// TwinCAT 3 PLC project Tc3_Element
// Title: Tc3_Element
// Company: Zerlauth
// Author: Peter Zerlauth
// ProjectVersion: 0.0.0.1
// Description: State Model with Observer and Events
// ProgramVersion: 3.1.4026.14
// CompilerDefines: release
// libraries:
//   Tc2_Standard, * (Beckhoff Automation GmbH)
//   Tc2_System, * (Beckhoff Automation GmbH)
//   Tc2_Utilities, * (Beckhoff Automation GmbH)
//   Tc3_Module,3.4.5.0,Beckhoff Automation GmbH
// project tree:
//   Element/Event/ E_Event.TcDUT, FB_Event.TcPOU, I_Event.TcIO, ST_Event.TcDUT (not stored), ST_EventFlags.TcDUT (not stored)
//   Element/Event/Observer/ FB_Observable.TcPOU (not stored), I_Observer.TcIO (not stored), I_Observable.TcIO (not stored)
//   Element/ E_Request.TcDUT, E_State.TcDUT, FB_Element.TcPOU, I_Element.TcIO (not stored)
//   Element/Reflection/ FB_Reflection.TcPOU (not stored), I_Reflection.TcIO
//   Element/Sequence/ E_Sequence.TcDUT (not stored), FB_Sequence.TcPOU (not stored), I_Sequence.TcIO (not stored), ST_Sequence.TcDUT (not stored), ST_SequenceOptions.TcDUT (not stored)
//   Level/ FB_Level.TcPOU
//   List/ FB_ListElement.TcPOU (not stored), FB_ListObject.TcPOU (not stored), FB_ListString.TcPOU (not stored), I_ListBase.TcIO (not stored), I_ListElement.TcIO (not stored), I_ListObject.TcIO (not stored), I_ListString.TcIO (not stored)
//   Logger/ FB_FileLogger.TcPOU, FB_LoggingProvider.TcPOU (not stored), FB_Logger.TcPOU, I_Logger.TcIO (not stored)
//   Module/ E_Mode.TcDUT (not stored), FB_Module.TcPOU, I_Module.TcIO (not stored)
//   Object/ FB_Object.TcPOU (not stored), I_Object.TcIO (not stored)
//   Utils/ FB_Debounce.TcPOU (not stored)
//   Utils/File/ FB_File.TcPOU, I_File.TcIO (not stored)
//   Version/ Global_Version.TcGVL (not stored)
// (motion and I/O tree: see PLC project development)
// real-time tasks:
//   TASK PlcTask: cycle T#500ms, priority 21, ADS port 351
//   TASK UnitTestTask: cycle T#1ms, priority 1, ADS port 350
// variable links:

// ---- Element/Event/E_Event.TcDUT
{attribute 'qualified_only'}
{attribute 'strict'}
{attribute 'to_string'}
TYPE E_Event :
(
	Verbose			:= 0,
	Debug			:= 1,
	Information		:= 2,
	Warning			:= 3,
	Error			:= 4
);
END_TYPE

// ---- Element/E_Request.TcDUT
{attribute 'qualified_only'}
{attribute 'strict'}
{attribute 'to_string'}

TYPE E_Request :
(
	{attribute 'analysis' := '-27'}
	Reset       := 1,
	{attribute 'analysis' := '-27'}
    Start       := 2,
	{attribute 'analysis' := '-27'}
	Stop		:= 3,
	{attribute 'analysis' := '-27'}
	Abort		:= 4
);
END_TYPE

// ---- Element/E_State.TcDUT
{attribute 'qualified_only'}
{attribute 'strict'}
{attribute 'to_string'}
TYPE E_State :
(
    Resetting       := 0,
   	Idle            := 1,
    Starting        := 2,
    Execute         := 3,
    Stopping        := 4,
    Stopped         := 5,
    Aborting        := 6,
    Aborted         := 7

)INT;
END_TYPE

// ---- Element/Event/I_Event.TcIO
INTERFACE I_Event EXTENDS I_Object

METHOD PUBLIC M_AddBOOL : I_Event
VAR_INPUT
	Value: 	BOOL;
END_VAR
END_METHOD

METHOD PUBLIC M_AddINT : I_Event
VAR_INPUT
	Value: 	LINT;
END_VAR
END_METHOD

METHOD PUBLIC M_AddREAL : I_Event
VAR_INPUT
	Value: 	Lreal;
	Decimals: INT;
END_VAR
END_METHOD

METHOD PUBLIC M_AddSTRING : I_Event
VAR_INPUT
	Value: STRING(255);
END_VAR
END_METHOD

METHOD PUBLIC M_AddTIME : I_Event
VAR_INPUT
	Value: 	TIME;
END_VAR
END_METHOD

METHOD PUBLIC M_Debug
VAR_INPUT
	sMessage:				STRING(255);
END_VAR
END_METHOD

METHOD PUBLIC M_Error
VAR_INPUT
	sMessage:				STRING(255);
	nID:					ULINT;
END_VAR
END_METHOD

METHOD PUBLIC M_Fatal
VAR_INPUT
	sMessage:				STRING(255);
	nID:					ULINT;
END_VAR
END_METHOD

METHOD PUBLIC M_Info
VAR_INPUT
	sMessage:				STRING(255);
	nID:					ULINT;
END_VAR
END_METHOD

METHOD PUBLIC M_Warning
VAR_INPUT
	sMessage:				STRING(255);
	nID:					ULINT;
END_VAR
END_METHOD

{attribute 'OPC.UA.DA.Property' := '1'}
{attribute 'monitoring' := 'call'}
PROPERTY PUBLIC P_Logger : I_Logger
GET
END_GET
SET
END_SET
END_PROPERTY

{attribute 'OPC.UA.DA.Property' := '1'}
{attribute 'monitoring' := 'call'}
PROPERTY PUBLIC P_Observer : I_Observable
GET
END_GET
END_PROPERTY

END_INTERFACE

// ---- Element/Reflection/I_Reflection.TcIO
INTERFACE I_Reflection

{attribute 'OPC.UA.DA.Property' := '1'}
{attribute 'monitoring' := 'call'}
PROPERTY PUBLIC P_Class : STRING(255)
GET
END_GET
END_PROPERTY

{attribute 'OPC.UA.DA.Property' := '1'}
{attribute 'monitoring' := 'call'}
PROPERTY PUBLIC P_Comment : STRING(255)
GET
END_GET
END_PROPERTY

{attribute 'OPC.UA.DA.Property' := '1'}
{attribute 'monitoring' := 'call'}
PROPERTY PUBLIC P_ID : STRING(25)
GET
END_GET
SET
END_SET
END_PROPERTY

{attribute 'OPC.UA.DA.Property' := '1'}
{attribute 'monitoring' := 'call'}
PROPERTY PUBLIC P_Instance : STRING(255)
GET
END_GET
END_PROPERTY

{attribute 'OPC.UA.DA.Property' := '1'}
{attribute 'monitoring' := 'call'}
PROPERTY PUBLIC P_Timestamp : DT
GET
END_GET
END_PROPERTY

END_INTERFACE

// ---- Element/Event/FB_Event.TcPOU
FUNCTION_BLOCK FB_Event IMPLEMENTS I_Event
VAR_INPUT
	fbObserver:			FB_Observable;				// Observer
END_VAR
VAR_OUTPUT
END_VAR
VAR
	{IF (defined (release))}
    	{attribute 'hide'}
	{END_IF}
	iLogger:			I_Logger;					// Event logger
	{IF (defined (release))}
    	{attribute 'hide'}
	{END_IF}
	iParent:			I_Element;					// Parent component
	{IF (defined (release))}
    	{attribute 'hide'}
	{END_IF}
	fbList:				FB_ListString;				// contains a list with string values
	stDebug:			ST_Event;					// last debug event
	stInfo:				ST_Event;					// last info event
	stWarning:			ST_Event;					// last warning event
	stError:			ST_Event;					// last error event
	stFatal:			ST_Event;					// last fatal event
END_VAR

// https://peterzerlauth.com/
fbObserver();

METHOD FB_init : BOOL
VAR_INPUT
	bInitRetains : BOOL; // if TRUE, the retain variables are initialized (warm start / cold start)
	bInCopyCode : BOOL;  // if TRUE, the instance afterwards gets moved into the copy code (online change)
	iParent:			I_Element;
END_VAR
THIS^.iParent:= iParent;
fbObserver.iParent:= iParent;
END_METHOD

METHOD PUBLIC M_AddBOOL : I_Event
VAR_INPUT
	Value: 	bool;
END_VAR
fbList.M_Add(BOOL_TO_STRING(Value));
M_AddBOOL:= THIS^;
END_METHOD

METHOD PUBLIC M_AddINT : I_Event
VAR_INPUT
	Value: 	LINT;
END_VAR
fbList.M_Add(LINT_TO_STRING(Value));
M_AddINT:= THIS^;
END_METHOD

METHOD PUBLIC M_AddREAL : I_Event
VAR_INPUT
	Value: 	Lreal;
	Decimals: INT;
END_VAR
fbList.M_Add(LREAL_TO_FMTSTR(Value, Decimals, TRUE));
M_AddREAL:= THIS^;
END_METHOD

METHOD PUBLIC M_AddSTRING : I_Event
VAR_INPUT
	Value: STRING(255);
END_VAR
fbList.M_Add(Value);
M_AddSTRING:= THIS^;
END_METHOD

METHOD PUBLIC M_AddTIME : I_Event
VAR_INPUT
	Value: 	TIME;
END_VAR
fbList.M_Add(TIME_TO_STRING(Value));
M_AddTIME:= THIS^;
END_METHOD

METHOD INTERNAL M_Arguments : STRING(255)
VAR_INPUT
END_VAR
VAR
	nIndex:			INT;
END_VAR
WHILE nIndex < fbList. P_Length DO
	M_Arguments:= Concat(Concat(M_Arguments, fbList.M_Index(nIndex)), '$N');
	nIndex:= nIndex + 1;
END_WHILE

fbList.M_Clear();
END_METHOD

METHOD INTERNAL M_Build : STRING(255)
VAR_INPUT
	sMessage:		STRING(255);
END_VAR
VAR
	nIndex:		   	DINT;
	nPosition: 		INT;
END_VAR
nPosition:= Find(sMessage, '%s');
WHILE nPosition <> 0 DO
	sMessage:= Replace(sMessage, fbList.M_Index(nIndex), 2, nPosition);
	nPosition:= Find(sMessage, '%s');
	nIndex:= nIndex + 1;
END_WHILE
M_Build:= sMessage;
END_METHOD

METHOD PUBLIC M_Debug
VAR_INPUT
	sMessage:				STRING(255);
END_VAR
stDebug.sMessage:= sMessage;
stDebug.iSource:= iParent;
stDebug.sInstance:= iParent.P_Reflection.P_Instance;
stDebug.sClass:= iParent.P_Reflection.P_Class;
stDebug.eEventType:= E_Event.Debug;
stDebug.tTimestamp:= iParent.P_Reflection.P_Timestamp;
stDebug.nID:= 0;
stDebug.sDefault:= M_Build(sMessage);
stDebug.sArguments:= M_Arguments();
stDebug.stFlags.bActive:= TRUE;
stDebug.stFlags.bRemove:= TRUE;

IF iLogger = 0 THEN
	M_Log(stDebug);
ELSE
	iLogger.M_Log(stDebug);
END_IF
END_METHOD

METHOD PUBLIC M_Error
VAR_INPUT
	sMessage:				STRING(255);
	nID:					ULINT;
END_VAR
stError.sMessage:= sMessage;
stError.iSource:= iParent;
stError.sInstance:= iParent.P_Reflection.P_Instance;
stError.sClass:= iParent.P_Reflection.P_Class;
stError.eEventType:= E_Event.Error;
stError.tTimestamp:= iParent.P_Reflection.P_Timestamp;
stError.nID:= nID;
stError.sDefault:= M_Build(sMessage);
stError.sArguments:= M_Arguments();
stError.stFlags.bActive:= TRUE;
stError.stFlags.bRemove:= TRUE;

IF iLogger = 0 THEN
	M_Log(stError);
ELSE
	iLogger.M_Log(stError);
END_IF
END_METHOD

METHOD PUBLIC M_Fatal
VAR_INPUT
	sMessage:				STRING(255);
	nID:					ULINT;
END_VAR
stFatal.sMessage:= sMessage;
stFatal.iSource:= iParent;
stFatal.sInstance:= iParent.P_Reflection.P_Instance;
stFatal.sClass:= iParent.P_Reflection.P_Class;
stFatal.eEventType:= E_Event.Error;
stFatal.tTimestamp:= iParent.P_Reflection.P_Timestamp;
stFatal.nID:= nID;
stFatal.sDefault:= M_Build(sMessage);
stFatal.sArguments:= M_Arguments();
stFatal.stFlags.bActive:= TRUE;
stFatal.stFlags.bRemove:= FALSE;

IF iLogger = 0 THEN
	M_Log(stFatal);
ELSE
	iLogger.M_Log(stFatal);
END_IF

fbObserver.M_Notify(iParent);
END_METHOD

METHOD PUBLIC M_Info
VAR_INPUT
	sMessage:				STRING(255);
	nID:					ULINT;
END_VAR
stInfo.sMessage:= sMessage;
stInfo.iSource:= iParent;
stInfo.sInstance:= iParent.P_Reflection.P_Instance;
stInfo.sClass:= iParent.P_Reflection.P_Class;
stInfo.eEventType:= E_Event.Information;
stInfo.tTimestamp:= iParent.P_Reflection.P_Timestamp;
stInfo.nID:= nID;
stInfo.sDefault:= M_Build(sMessage);
stInfo.sArguments:= M_Arguments();
stInfo.stFlags.bActive:= TRUE;
stInfo.stFlags.bRemove:= TRUE;

IF iLogger = 0 THEN
	M_Log(stInfo);
ELSE
	iLogger.M_Log(stInfo);
END_IF
END_METHOD

METHOD PRIVATE M_Log : BOOL
VAR_INPUT
	stEvent	: ST_Event;
END_VAR
// @ToDo
END_METHOD

METHOD PUBLIC M_Warning
VAR_INPUT
	sMessage:				STRING(255);
	nID:					ULINT;
END_VAR
stWarning.sMessage:= sMessage;
stWarning.iSource:= iParent;
stWarning.sInstance:= iParent.P_Reflection.P_Instance;
stWarning.sClass:= iParent.P_Reflection.P_Class;
stWarning.eEventType:= E_Event.Warning;
stWarning.tTimestamp:= iParent.P_Reflection.P_Timestamp;
stWarning.nID:= nID;
stWarning.sDefault:= M_Build(sMessage);
stWarning.sArguments:= M_Arguments();
stWarning.stFlags.bActive:= TRUE;
stWarning.stFlags.bRemove:= TRUE;

IF iLogger = 0 THEN
	M_Log(stWarning);
ELSE
	iLogger.M_Log(stWarning);
END_IF
END_METHOD

{attribute 'OPC.UA.DA.Property' := '1'}
{attribute 'monitoring' := 'call'}
PROPERTY P_Logger : I_Logger
GET
P_Logger:= iLogger;
END_GET
SET
iLogger:= P_Logger;
END_SET
END_PROPERTY

{attribute 'OPC.UA.DA.Property' := '1'}
{attribute 'monitoring' := 'call'}
PROPERTY PUBLIC P_Observer : I_Observable
GET
P_Observer:= fbObserver;
END_GET
END_PROPERTY

END_FUNCTION_BLOCK

// ---- Element/FB_Element.TcPOU
FUNCTION_BLOCK FB_Element IMPLEMENTS I_Element
VAR_INPUT
END_VAR
VAR_OUTPUT
END_VAR
VAR
	fbReflection:					FB_Reflection;				// Info about function block
	fbEvent:						FB_Event(THIS^);			// Event Publisher
	fbSequence:						FB_Sequence(THIS^);			// Sequence
	{attribute 'OPC.UA.DA' := '1'}
	{attribute 'OPC.UA.DA.Access' := '2'}
	eState:							E_State;					// Current state
	{attribute 'OPC.UA.DA' := '1'}
	{attribute 'OPC.UA.DA.Access' := '1'}
	eStateRequest:					E_State;					// State command
    {attribute 'hide'}
	eStatePrevious:					E_State;					// Previous state
END_VAR

fbReflection();
fbEvent();
fbSequence();

// State machine logic
CASE eState OF

    // Idle state:
    E_State.Idle:
        IF M_Idle() THEN
            eState := E_State.Starting;
        END_IF
		
		CASE eStateRequest OF
			E_State.Starting, E_State.Execute:
            	eState := E_State.Starting;
	
			E_State.Stopping, E_State.Stopped:
            	eState := E_State.Stopping;

			E_State.Aborting, E_State.Aborted:
            	eState := E_State.Aborting;
	
		END_CASE

    // Starting state:
    E_State.Starting:
        IF M_Starting() THEN
            eState := E_State.Execute;
        END_IF
		
		CASE eStateRequest OF
			E_State.Stopping, E_State.Stopped:
            	eState := E_State.Stopping;

			E_State.Aborting, E_State.Aborted:
            	eState := E_State.Aborting;
	
		END_CASE
			
    // Execute state:
    E_State.Execute:
        IF M_Execute() THEN
            eState := E_State.Stopping;
        END_IF
		
		CASE eStateRequest OF
			E_State.Stopping, E_State.Stopped:
            	eState := E_State.Stopping;

			E_State.Aborting, E_State.Aborted:
            	eState := E_State.Aborting;				

		END_CASE

    // Stopping state:
    E_State.Stopping:
        IF M_Stopping() THEN
            eState := E_State.Stopped;
        END_IF
		CASE eStateRequest OF
			E_State.Aborting, E_State.Aborted:
            	eState := E_State.Aborting;				

		END_CASE

    // Stopped state:
    E_State.Stopped:
        IF M_Stopped() THEN
            eState := E_State.Resetting;
        END_IF
		
		CASE eStateRequest OF
			E_State.Resetting, E_State.Idle:
            eState := E_State.Resetting;			
			
		END_CASE
		
    // Aborting state:
    E_State.Aborting:
        IF M_Aborting() THEN
            eState := E_State.Aborted;
        END_IF

    // Aborted state:
    E_State.Aborted:
        IF M_Aborted() THEN
            eState := E_State.Resetting;
        END_IF
		
		CASE eStateRequest OF
			E_State.Resetting, E_State.Idle:
            eState := E_State.Resetting;			
			
		END_CASE

    // Resetting state:
    E_State.Resetting:
        IF M_Resetting() THEN
            eState := E_State.Idle;
        END_IF

END_CASE
eStateRequest := eState;

// Detect state transitions and trigger event callback
IF eStatePrevious <> eState THEN
    M_OnState(eState, eStatePrevious);
    eStatePrevious := eState;
END_IF

METHOD PROTECTED M_Aborted : BOOL // Return
VAR_INPUT
END_VAR
M_Aborted:= FALSE;
END_METHOD

METHOD PROTECTED M_Aborting : BOOL // Return
VAR_INPUT
END_VAR
M_Aborting:= TRUE;
END_METHOD

METHOD PROTECTED M_Completed : BOOL // Return
VAR_INPUT
END_VAR
M_Completed:= TRUE;
END_METHOD

METHOD PROTECTED M_Completing : BOOL // Return
VAR_INPUT
END_VAR
M_Completing:= TRUE;
END_METHOD

METHOD PROTECTED M_Execute : BOOL // Return
VAR_INPUT
END_VAR
M_Execute:= FALSE;
END_METHOD

METHOD PROTECTED M_Idle : BOOL // Return
VAR_INPUT
END_VAR
M_Idle:= FALSE;
END_METHOD

METHOD Protected M_OnState
VAR_INPUT
	eState:							E_State;						// Current state
	eStatePrevious:					E_State;						// Previous state	
END_VAR
// State changed event
fbSequence.M_Reset();
END_METHOD

{attribute 'TcRpcEnable':='1'}
METHOD PUBLIC M_Request : BOOL
VAR_INPUT
	eRequest:	E_Request;
END_VAR
// Request element states
CASE eRequest OF
	E_Request.Reset:
		eStateRequest:= E_State.Resetting;
		CASE eState OF
			E_State.Execute, E_State.Idle:
				M_Request:= TRUE;
		END_CASE

	E_Request.Start:
		eStateRequest:= E_State.Execute;
		CASE eState OF 
			E_State.Execute:
				M_Request:= TRUE;
		END_CASE

	E_Request.Stop:
		eStateRequest:= E_State.Stopped;
		CASE eState OF
			E_State.Stopped, E_State.Aborted, E_State.Idle:
				M_Request:= TRUE;
		END_CASE

	E_Request.Abort:
		eStateRequest:= E_State.Aborted;
		CASE eState OF
			E_State.Aborted:
				M_Request:= TRUE;
		END_CASE	

END_CASE
END_METHOD

METHOD PROTECTED M_Resetting : BOOL // Return
VAR_INPUT
END_VAR
M_Resetting:= TRUE;
END_METHOD

METHOD PROTECTED M_Starting : BOOL // Return
VAR_INPUT
END_VAR
M_Starting:= TRUE;
END_METHOD

METHOD PROTECTED M_Stopped : BOOL // Return
VAR_INPUT
END_VAR
M_Stopped:= FALSE;
END_METHOD

METHOD PROTECTED M_Stopping : BOOL // Return state complete
VAR_INPUT
END_VAR
M_Stopping:= TRUE;
END_METHOD

PROPERTY PUBLIC P_Event : I_Event
GET
P_Event:= fbEvent;
END_GET
END_PROPERTY

PROPERTY PUBLIC P_Reflection : I_Reflection
GET
P_Reflection:= fbReflection;
END_GET
END_PROPERTY

PROPERTY PUBLIC P_Sequence : I_Sequence
GET
P_Sequence:= fbSequence;
END_GET
END_PROPERTY

PROPERTY PUBLIC P_State : E_State
GET
P_State:= eState;
END_GET
END_PROPERTY

END_FUNCTION_BLOCK

// ---- Level/FB_Level.TcPOU
FUNCTION_BLOCK FB_Level EXTENDS FB_Element
VAR_INPUT
	fbList:				FB_ListElement;
END_VAR
VAR_OUTPUT
END_VAR
VAR
END_VAR

SUPER^();

METHOD PROTECTED M_Aborting : BOOL (* Return*)
VAR
	nIndex: 	UINT;
END_VAR
M_Aborting:= TRUE;
WHILE nIndex < fbList.nLength DO
    IF fbList.M_Index(nIndex).M_Request(E_Request.Abort) THEN
		;
	ELSE
		M_Aborting:= FALSE;
	END_IF
	nIndex := nIndex + 1;
END_WHILE
END_METHOD

METHOD PUBLIC M_Attach : BOOL
VAR_INPUT
	iComponent:		I_Element;
END_VAR
fbList.M_Add(iComponent);
iComponent.P_Event.P_Logger:= fbEvent.P_Logger;
iComponent.P_Event.P_Observer.M_Attach(THIS^);
fbEvent.fbObserver.M_Attach(iComponent);
M_Attach:= TRUE;
END_METHOD

METHOD PUBLIC M_Detach : BOOL
VAR_INPUT
END_VAR
END_METHOD

METHOD PROTECTED M_Resetting : BOOL (* Return*)
VAR
	nIndex: 	UINT;
END_VAR
M_Resetting:= TRUE;
WHILE nIndex < fbList.nLength DO
    IF fbList.M_Index(nIndex).M_Request(E_Request.Reset) THEN
		;
	ELSE
		M_Resetting:= FALSE;
	END_IF
	nIndex := nIndex + 1;
END_WHILE
END_METHOD

METHOD PROTECTED M_Starting : BOOL (* Return*)
VAR
	nIndex: 	UINT;
END_VAR
M_Starting:= TRUE;
WHILE nIndex < fbList.nLength DO
    IF fbList.M_Index(nIndex).M_Request(E_Request.Start) THEN
		;
	ELSE
		M_Starting:= FALSE;
	END_IF
	nIndex := nIndex + 1;
END_WHILE
END_METHOD

METHOD PROTECTED M_Stopping : BOOL (* Return state complete*)
VAR
	nIndex: 	UINT;
END_VAR
M_Stopping:= TRUE;
WHILE nIndex < fbList.nLength DO
    IF fbList.M_Index(nIndex).M_Request(E_Request.Reset) THEN
		;
	ELSE
		M_Stopping:= FALSE;
	END_IF
	nIndex := nIndex + 1;
END_WHILE
END_METHOD

PROPERTY PUBLIC P_List : I_ListElement
GET
P_List:= fbList;
END_GET
END_PROPERTY

END_FUNCTION_BLOCK

// ---- Logger/FB_FileLogger.TcPOU
FUNCTION_BLOCK FB_FileLogger VAR_GENERIC CONSTANT nMaxLength: UINT := 10; END_VAR IMPLEMENTS I_Logger
VAR_INPUT
	sPathName:					STRING;
END_VAR
VAR
	nLength:					DINT;
	aEvent:						ARRAY [0..nMaxLength - 1] OF ST_Event;
	fbFile:						FB_File;
	bWriteLine:					BOOL;
	bOpen:						BOOL;
	bClose: 					BOOL;
END_VAR

// https://peterzerlauth.com/

fbFile();

IF bOpen THEN
	bOpen:= NOT fbFile.M_Open(sPathName);
END_IF

IF bWriteLine THEN
	bWriteLine:= NOT fbFile.M_AppendLine('Test');
END_IF


IF bClose THEN
	bClose:= NOT fbFile.M_Close();
END_IF

METHOD PUBLIC M_Delete : BOOL
VAR_INPUT
	nIndex: 			DINT;
END_VAR
// new Length
nLength:= nLength -1;
//pList[nPosition]:= iObject;
Memcpy(ADR(aEvent[nIndex]), ADR(aEvent[nIndex +1]), SIZEOF(POINTER TO ST_Event) * DINT_TO_UDINT(nMaxLength - nIndex));
END_METHOD

METHOD PUBLIC M_Find : DINT
VAR_INPUT
	stEvent:	ST_Event;
END_VAR
VAR 
	nIndex:		DINT;
END_VAR
// Find event in buffer
M_Find := -1;
WHILE nIndex < nLength DO
	IF (aEvent[nIndex].iSource = stEvent.iSource) AND_THEN
    	(aEvent[nIndex].eEventType = stEvent.eEventType) AND_THEN
		(aEvent[nIndex].sInstance = stEvent.sInstance) AND_THEN
		(aEvent[nIndex].sMessage = stEvent.sMessage) THEN
        M_Find := nIndex;
        RETURN;
    END_IF
	nIndex := nIndex + 1;
END_WHILE
END_METHOD

METHOD PUBLIC M_Log
VAR_INPUT
	stEvent:		ST_Event;
END_VAR
VAR
	nIndex:			DINT;
END_VAR
IF (nIndex:=  M_Find(stEvent)) >= 0 THEN
	// Update existing events
	aEvent[nIndex].sArguments:= stEvent.sArguments;
	aEvent[nIndex].sDefault:= stEvent.sDefault;
	aEvent[nIndex].sClass:= stEvent.sClass;
	aEvent[nIndex].stFlags:= stEvent.stFlags;
	
ELSE
	// add new event
	aEvent[nLength]:= stEvent;
	nLength:= nLength + 1;
	
// 	fbFile.M_AppendLine(stEvent.eEventType
END_IF
END_METHOD

METHOD PUBLIC M_Reset
VAR_INPUT
END_VAR
// Reset all events
nLength:= 0;
Memset(ADR(aEvent), 0, SIZEOF(aEvent));
END_METHOD

END_FUNCTION_BLOCK

// ---- Utils/File/FB_File.TcPOU
{attribute 'no_explicit_call'} 
FUNCTION_BLOCK FB_File
VAR
    fbCreateDir:	FB_CreateDir;
	fbOpen:			FB_FileOpen;
	fbRead:			FB_FileRead;
	fbLoad:			FB_FileLoad;
	fbPuts:			FB_FilePuts;
	fbWrite:		FB_FileWrite;
	fbClose:		FB_FileClose;
	fbDelete:		FB_FileDelete;
END_VAR
VAR_INPUT
	nMode:			DWORD:= (FOPEN_MODEAPPEND OR FOPEN_MODEPLUS OR FOPEN_MODETEXT);
END_VAR
VAR_OUTPUT
	nError:			UDINT;
END_VAR

// https://peterzerlauth.com/
fbCreateDir();
fbLoad();
fbOpen();
fbDelete();
fbPuts();
fbWrite();
fbRead();
fbClose();

METHOD PUBLIC M_Append : BOOL
VAR_INPUT
	Text:			T_MaxString;
END_VAR
IF fbPuts.bExecute THEN
	IF fbPuts.bError THEN
		nError:= fbPuts.nErrId;
		fbPuts.bExecute:= FALSE;
	ELSIF fbPuts.bBusy THEN
		;
	ELSE
		M_Append:= TRUE;
		fbPuts.bExecute:= FALSE;
	END_IF
ELSE
	fbPuts.bExecute:= TRUE;
	fbPuts.sLine:= Text;
END_IF
END_METHOD

METHOD PUBLIC M_AppendLine : BOOL
VAR_INPUT
	Line:			T_MaxString;
END_VAR
IF fbPuts.bExecute THEN
	IF fbPuts.bError THEN
		nError:= fbPuts.nErrId;
		fbPuts.bExecute:= FALSE;
	ELSIF fbPuts.bBusy THEN
		;
	ELSE
		M_AppendLine:= TRUE;
		fbPuts.bExecute:= FALSE;
	END_IF
ELSE
	fbPuts.bExecute:= TRUE;
	fbPuts.sLine:= Concat(Line, '$R');
END_IF
END_METHOD

METHOD PUBLIC M_Close : BOOL
VAR_INPUT
END_VAR
IF fbClose.bExecute THEN
	IF fbClose.hFile = 0 THEN
		fbClose.bExecute:= FALSE;
		M_Close:= TRUE;
	ELSIF fbClose.bError THEN
		fbClose.bExecute:= FALSE;
		nError:= fbClose.nErrId;
	ELSIF fbClose.bBusy THEN
		;
	ELSE
		nError:= 0;	
		fbRead.hFile:= 0;
		fbPuts.hFile:= 0;
		fbWrite.hFile:= 0;
		fbClose.hFile:= 0;
		fbClose.bExecute:= FALSE;
		M_Close:= TRUE;
	END_IF
ELSE
	fbClose.bExecute:= TRUE;
END_IF
END_METHOD

METHOD PUBLIC M_Create : BOOL
VAR_INPUT
	PathName:		STRING(255);
END_VAR
VAR
	nTemp: INT;
END_VAR
VAR_INST
	nPosition: INT;
END_VAR
nTemp := FIND(RIGHT(PathName, LEN(PathName) - nPosition), '\');
if nTemp <> 0 then
	IF fbCreateDir.bExecute THEN
		IF NOT fbCreateDir.bBusy THEN
			nPosition := nPosition + nTemp;
			fbCreateDir.bExecute:= FALSE;
		END_IF
	ELSE
		fbCreateDir.bExecute:= TRUE;
		fbCreateDir.ePath:= PATH_GENERIC;
		fbCreateDir.sPathName:= Left(PathName, nPosition + nTemp);
	END_IF
ELSE
	IF M_Open(PathName) THEN
		M_Create:= TRUE;
		nPosition:= 0;
	END_IF
END_IF
END_METHOD

METHOD PUBLIC M_Delete : BOOL
VAR_INPUT
	PathName:		STRING(255);
END_VAR
IF fbDelete.bExecute THEN
	IF fbDelete.bError THEN
		fbDelete.bExecute:= FALSE;
		M_Delete:= TRUE;
	ELSIF fbDelete.bBusy THEN
		;
	ELSE
		fbDelete.bExecute:= FALSE;
		M_Delete:= TRUE;
	END_IF
ELSE
	fbDelete.bExecute:= TRUE;
	fbDelete.sPathName:= PathName;
	fbDelete.ePath:= E_OpenPath.PATH_GENERIC;
END_IF
END_METHOD

METHOD PUBLIC M_Load : BOOL
VAR_INPUT
	PathName:		STRING(255);
	Value:			ANY;
END_VAR
IF fbLoad.bExecute THEN
	IF fbLoad.bError THEN
		nError:= fbLoad.nErrId;
		fbLoad.bExecute:= FALSE;
	ELSIF fbLoad.bBusy THEN
		;
	ELSE
		M_Load:= TRUE;
	END_IF
ELSE
	fbLoad.sPathName:= PathName;
	fbLoad.bExecute:= TRUE;
	fbLoad.pReadBuff:= Value.pValue;
	fbLoad.cbReadLen:= DINT_TO_UDINT(Value.diSize);
END_IF
END_METHOD

METHOD PUBLIC M_Open : BOOL
VAR_INPUT
	PathName:		STRING(255);
END_VAR
// Check if the file open should be executed
IF fbOpen.bExecute THEN
    // Check the file opening process
    IF fbOpen.bError THEN
        // Store the error ID and stop the execution
        nError:= fbOpen.nErrId;
        fbOpen.bExecute:= FALSE;
        
    // If the process is still busy, do nothing and wait
    ELSIF fbOpen.bBusy THEN
        ;
    // If the file has been successfully opened
    ELSE
        fbOpen.bExecute:= FALSE;
    END_IF    
ELSE
    // If the file handle is invalid (e.g., the file is not open)
    IF fbOpen.hFile <> 0 THEN
		// Assign the file handle
		fbRead.hFile:= fbOpen.hFile;
		fbPuts.hFile:= fbOpen.hFile;
        fbWrite.hFile:= fbOpen.hFile;
        fbClose.hFile:= fbOpen.hFile;
		 // file is open
        M_Open:= TRUE;    
    ELSE
        // Start the file opening process with the specified path and mode
        fbOpen.bExecute:= TRUE;
        fbOpen.sPathName:= PathName;
        fbOpen.nMode:= nMode;   
    END_IF
END_IF
END_METHOD

METHOD PUBLIC M_Read : BOOL
VAR_INPUT
	Value:		ANY;
END_VAR
IF fbRead.bExecute THEN
	IF fbRead.bError THEN
		nError:= fbRead.nErrId;
		fbRead.bExecute:= FALSE;
	ELSIF fbRead.bBusy THEN
		;
	ELSE
		fbRead.bExecute:= FALSE;
		M_Read:= TRUE;
	END_IF
ELSE
	fbRead.bExecute:= TRUE;
	fbRead.pReadBuff:= Value.pValue;
	fbRead.cbReadLen:= DINT_TO_UDINT(Value.diSize);
END_IF
END_METHOD

METHOD PUBLIC M_Write : BOOL
VAR_INPUT
	Value:		ANY;
END_VAR
IF fbWrite.bExecute THEN
	IF fbWrite.bError THEN
		nError:= fbWrite.nErrId;
		fbWrite.bExecute:= FALSE;
	ELSIF fbWrite.bBusy THEN
		M_Write:= FALSE;
	ELSE
		M_Write:= TRUE;
		fbWrite.bExecute:= FALSE;
	END_IF
ELSE
	fbWrite.bExecute:= TRUE;
	fbWrite.pWriteBuff:= Value.pValue;
	fbWrite.cbWriteLen:= DINT_TO_UDINT(Value.diSize);
END_IF
END_METHOD

PROPERTY PUBLIC P_Error : UDINT
GET
P_Error:= nError;
END_GET
END_PROPERTY

PROPERTY PUBLIC P_Open : Bool
GET
P_Open:= fbOpen.hFile <> 0;
END_GET
END_PROPERTY

END_FUNCTION_BLOCK

// ---- Logger/FB_Logger.TcPOU
FUNCTION_BLOCK FB_Logger VAR_GENERIC CONSTANT nMaxLength: UINT := 10; END_VAR IMPLEMENTS I_Logger
VAR
	nLength:					DINT;
	aEvent:						ARRAY [0..nMaxLength - 1] OF ST_Event;
	nIndex: 					DINT;
	nTimestamp: 				ULINT;
END_VAR

// https://peterzerlauth.com/
// Execute each secound
IF nTimestamp <= F_GetSystemTime() THEN
	nTimestamp:= F_GetSystemTime() + 10000000;
	nIndex:= 0;
	WHILE nIndex < nLength DO
		IF aEvent[nIndex].stFlags.bActive THEN
			IF aEvent[nIndex].stFlags.bRemove THEN
				aEvent[nIndex].stFlags.bActive:= FALSE;
			END_IF
		ELSE
			M_Delete(nIndex);
		END_IF
		nIndex := nIndex + 1;
	END_WHILE
END_IF

METHOD PUBLIC M_Delete : BOOL
VAR_INPUT
	nIndex: 			DINT;
END_VAR
// new Length
nLength:= nLength -1;
MEMCPY(ADR(aEvent[nIndex]), ADR(aEvent[nIndex +1]), SIZEOF(ST_Event) * DINT_TO_UDINT(nMaxLength - nIndex));
END_METHOD

METHOD PUBLIC M_Find : DINT
VAR_INPUT
	stEvent:	ST_Event;
END_VAR
VAR 
	nIndex:		DINT;
END_VAR
// Find event in buffer
M_Find := -1;
WHILE nIndex < nLength DO
	IF (aEvent[nIndex].iSource = stEvent.iSource) AND_THEN
    	(aEvent[nIndex].eEventType = stEvent.eEventType) AND_THEN
		(aEvent[nIndex].sInstance = stEvent.sInstance) AND_THEN
		(aEvent[nIndex].sMessage = stEvent.sMessage) THEN
        M_Find := nIndex;
        RETURN;
    END_IF
	nIndex := nIndex + 1;
END_WHILE
END_METHOD

METHOD PUBLIC M_Log
VAR_INPUT
	stEvent:		ST_Event;
END_VAR
VAR
	nIndex:			DINT;
END_VAR
IF (nIndex:=  M_Find(stEvent)) >= 0 THEN
	// Update existing events
	aEvent[nIndex].sArguments:= stEvent.sArguments;
	aEvent[nIndex].sDefault:= stEvent.sDefault;
	aEvent[nIndex].sClass:= stEvent.sClass;
	aEvent[nIndex].stFlags:= stEvent.stFlags;
ELSE
	// add new event
	aEvent[nLength]:= stEvent;
	nLength:= nLength + 1;
END_IF
END_METHOD

METHOD PUBLIC M_Reset
VAR_INPUT
END_VAR
// Reset all events
nLength:= 0;
Memset(ADR(aEvent), 0, SIZEOF(aEvent));
END_METHOD

END_FUNCTION_BLOCK

// ---- Module/FB_Module.TcPOU
FUNCTION_BLOCK FB_Module EXTENDS FB_Element IMPLEMENTS I_Module
VAR_INPUT
END_VAR
VAR_OUTPUT
END_VAR
VAR
	{attribute 'OPC.UA.DA' := '1'}
	{attribute 'OPC.UA.DA.Access' := '2'}
	eMode:							E_Mode;							// Current mode
		{attribute 'OPC.UA.DA' := '1'}
	{attribute 'OPC.UA.DA.Access' := '1'}
	eModeRequest:					E_Mode:= E_Mode.Automatic;		// Requested mode
	{attribute 'hide'}
	eModePrevious:					E_Mode;							// Previous mode
	
	fbLogging:					FB_LoggingProvider;
	fbLogger:					FB_Logger<20>;
	
	fbLevel1:					FB_Level;
	fbLevel2:					FB_Level;
	fbLevel3:					FB_Level;
	fbLevel4:					FB_Level;
END_VAR

// https://peterzerlauth.com/
SUPER^();

fbLogger();

fbLevel1();
fbLevel2();
fbLevel3();
fbLevel4();

// Detect mode changes
IF eModeRequest <> E_Mode.Undefined THEN
	IF eMode <> eModeRequest THEN
		eModePrevious:= eMode;
		eMode:= eModeRequest;
		M_OnMode(eMode, eModePrevious);
	END_IF
END_IF
eModeRequest:= E_Mode.Undefined;

METHOD PROTECTED M_Aborting : BOOL (* Return*)
M_Aborting:= 	fbLevel4.M_Request(E_Request.Abort) AND
 				fbLevel3.M_Request(E_Request.Abort) AND
				fbLevel2.M_Request(E_Request.Abort) AND
				fbLevel1.M_Request(E_Request.Abort);
END_METHOD

METHOD PROTECTED M_Idle : BOOL (* Return*)
fbLogging.M_Add(fbLogger);

fbLevel4.P_Event.P_Logger:= fbLogging;
fbLevel3.P_Event.P_Logger:= fbLogging;
fbLevel2.P_Event.P_Logger:= fbLogging;
fbLevel1.P_Event.P_Logger:= fbLogging;

fbLevel4.P_Event.P_Observer.M_Attach(THIS^);
fbLevel3.P_Event.P_Observer.M_Attach(THIS^);
fbLevel2.P_Event.P_Observer.M_Attach(THIS^);
fbLevel1.P_Event.P_Observer.M_Attach(THIS^);

fbLevel4.M_Attach(fbLevel3);
fbLevel4.M_Attach(fbLevel2);
fbLevel4.M_Attach(fbLevel1);

fbLevel3.M_Attach(fbLevel2);
fbLevel3.M_Attach(fbLevel1);

fbLevel2.M_Attach(fbLevel1);

fbEvent.fbObserver.M_Attach(fbLevel1);
END_METHOD

{attribute 'TcRpcEnable':='1'}
METHOD PUBLIC M_Mode : BOOL
VAR_INPUT
	eMode:		E_Mode;
END_VAR
IF THIS^.eMode = eMode THEN
	M_Mode:= TRUE;
ELSE
	eModeRequest:= eMode;	
END_IF
END_METHOD

METHOD PROTECTED M_OnMode
VAR_INPUT
	eMode:							E_Mode;						// Current mode
	eModePrevious:					E_Mode;						// Previous mode	
END_VAR
CASE eMode OF
	E_Mode.Semiauto, E_Mode.Automatic:
		IF eModePrevious = E_Mode.Manual THEN
			fbEvent.M_AddSTRING(TO_STRING(eModePrevious));
			fbEvent.M_AddSTRING(TO_STRING(eMode));
			fbEvent.M_Fatal('Module mode changed form %s to %s', 1002);
		END_IF
	E_Mode.Manual:
		;
END_CASE
END_METHOD

METHOD PROTECTED M_Resetting : BOOL (* Return*)
M_Resetting:= 	fbLevel4.M_Request(E_Request.Reset) AND
 				fbLevel3.M_Request(E_Request.Reset) AND
				fbLevel2.M_Request(E_Request.Reset) AND
				fbLevel1.M_Request(E_Request.Reset);
END_METHOD

METHOD PROTECTED M_Starting : BOOL
VAR_INPUT
END_VAR
M_Starting:= 	fbLevel4.M_Request(E_Request.Start);
END_METHOD

METHOD PROTECTED M_Stopping : BOOL (* Return state complete*)
M_Stopping:= 	fbLevel3.M_Request(E_Request.Stop) AND
				fbLevel2.M_Request(E_Request.Stop) AND
				fbLevel1.M_Request(E_Request.Stop);
END_METHOD

PROPERTY PUBLIC P_Mode : E_Mode
GET
P_Mode:= eMode;
END_GET
END_PROPERTY

END_FUNCTION_BLOCK
